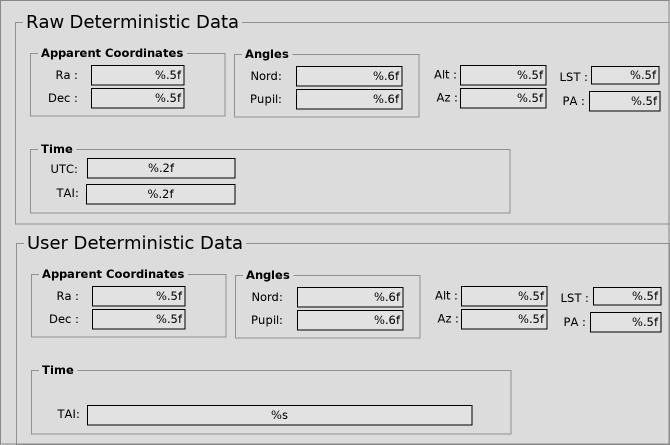
VISUALIZATION GUI_TEMPLATE_CCS_RECEIVER  // 670x445
VAR_INPUT
	m_DeviceName : STRING;
END_VAR
VAR_IN_OUT
	m_Instance : FB_CCS_SIM;
END_VAR
    GroupBox (16,235 654x210), "User Deterministic Data"
        GroupBox (15,31 195x71), "Apparent Coordinates"
            Label (11,20 40x20), "Ra :"
            Label (11,43 40x20), "Dec :"
            Label (8,70 60x20)
            Rectangle (61,43 93x20), "%.5f", tooltip "Apparent Declination [ddmmss]", text variable: m_Instance.tracking_ccs.dec
            Rectangle (61,20 93x20), "%.5f", tooltip "Apparent Right Ascension [hhmmss]", text variable: m_Instance.tracking_ccs.ra
        Rectangle (574,77 71x20), "%.5f", tooltip "Parallactic Angle [deg]", text variable: m_Instance.tracking_ccs.pa
        Label (523,77 50x20), "PA :"
        Label (408,51 37x19), "Alt :"
        Label (411,74 35x19), "Az :"
        Rectangle (445,74 86x20), "%.5f", tooltip "TEL Azimuth [deg]", text variable: m_Instance.tracking_ccs.az
        Rectangle (445,51 86x20), "%.5f", tooltip "TEL Altitude [deg]", text variable: m_Instance.tracking_ccs.alt
        GroupBox (15,127 480x72), "Time"
            Label (6,42 46x20), "TAI:"
            Label (8,70 60x20)
            Rectangle (56,43 385x20), "%s", tooltip "TAI time", text variable: m_Instance.tracking_ccs.time_tai
        GroupBox (219,32 185x71), "Angles"
            Label (11,20 40x20), "Nord:"
            Label (11,43 40x20), "Pupil:"
            Label (8,70 60x20)
            Rectangle (62,20 106x20), "%.6f", tooltip "North angle [deg]", text variable: m_Instance.tracking_ccs.north_angle
            Rectangle (62,43 106x20), "%.6f", tooltip "Pupil angle[deg]", text variable: m_Instance.tracking_ccs.pupil_angle
        Label (534,53 42x20), "LST :"
    GroupBox (15,14 654x210), "Raw Deterministic Data"
        GroupBox (15,31 195x71), "Apparent Coordinates"
            Label (11,20 40x20), "Ra :"
            Label (11,43 40x20), "Dec :"
            Label (8,70 60x20)
            Rectangle (61,43 93x20), "%.5f", tooltip "Apparent Declination [rad]", text variable: m_Instance.tracking_raw.radec_at_altaz_at_requested_xy[1]
            Rectangle (61,20 93x20), "%.5f", tooltip "Apparent Right Ascension [rad]", text variable: m_Instance.tracking_raw.radec_at_altaz_at_requested_xy[0]
        Rectangle (574,77 71x20), "%.5f", tooltip "Parallactic Angle [rad]", text variable: m_Instance.tracking_raw.parallactic_angle
        Label (523,77 50x20), "PA :"
        Label (408,51 37x19), "Alt :"
        Label (411,74 35x19), "Az :"
        Rectangle (445,74 86x20), "%.5f", tooltip "TEL Azimuth [rad]", text variable: m_Instance.tracking_raw.current_observed_altaz[1]
        Rectangle (445,51 86x20), "%.5f", tooltip "TEL Altitude [rad]", text variable: m_Instance.tracking_raw.current_observed_altaz[0]
        GroupBox (15,127 480x72), "Time"
            Label (11,18 40x20), "UTC:"
            Label (6,42 46x20), "TAI:"
            Label (8,70 60x20)
            Rectangle (57,17 148x20), "%.2f", tooltip "UTC time [sec]", text variable: m_Instance.tracking_raw.time_utc
            Rectangle (56,43 149x20), "%.2f", tooltip "TAI time [sec]", text variable: m_Instance.tracking_raw.time_tai
        GroupBox (219,32 185x71), "Angles"
            Label (11,20 40x20), "Nord:"
            Label (11,43 40x20), "Pupil:"
            Label (8,70 60x20)
            Rectangle (62,20 106x20), "%.6f", tooltip "North angle [rad]", text variable: m_Instance.tracking_raw.north_angle
            Rectangle (62,43 106x20), "%.6f", tooltip "Pupil angle[rad]", text variable: m_Instance.tracking_raw.pupil_angle
        Label (534,53 42x20), "LST :"
        Rectangle (578,273 68x18), "%.5f", tooltip "Local Sidereal Time [h]", text variable: m_Instance.tracking_ccs.lst
    Rectangle (591,66 68x18), "%.5f", tooltip "Local Sidereal Time [h]", text variable: m_Instance.tracking_raw.time_lst
END_VISUALIZATION

(* stored: Version 1.1.0.1, ProductVersion 3.1.4024.11
   Visu GUI_TEMPLATE_CCS_RECEIVER: Id {f233d3d3-a08f-4bf9-918e-57222bcffbb9} *)
